% RSLogix 500 project vendingmachine.RSS, saved by version 9.00.00.04 %
PROJECT "UNTITLED"    % processor: MicroLogix 1200 %

PROGRAM FILES
  LAD 2   11 rungs

DATA FILES
  O0 OUTPUT  4 elements
  I1 INPUT  4 elements
  S2 STATUS  66 elements
  B3 BINARY  1 elements
  T4 TIMER  1 elements
  C5 COUNTER  1 elements
  R6 CONTROL  1 elements
  N7 INTEGER  1 elements
  F8 FLOAT  2 elements
  F9 PRICES  1 elements

LADDER 2
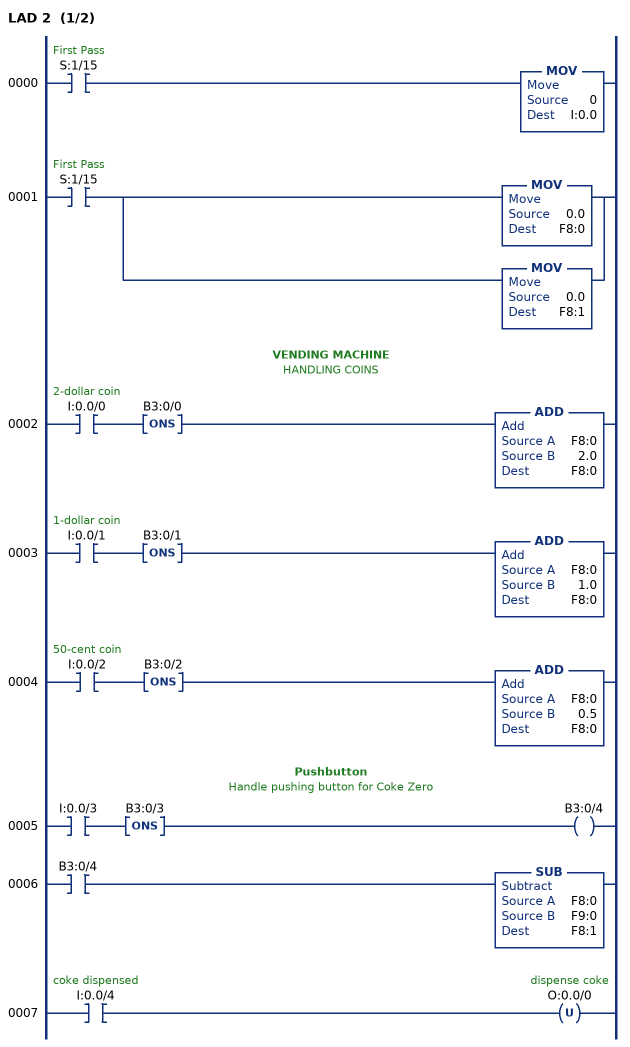
% Rung: 0 %
SOR XIC S:1/15 MOV 0 I:0.0 EOR
%   S:1/15  "First Pass" %
% Rung: 1 %
SOR XIC S:1/15 BST MOV 0.0 F8:0 NXB MOV 0.0 F8:1 BND EOR
%   S:1/15  "First Pass" %
% Rung: 2 %
% TITLE: VENDING MACHINE %
%                                                            HANDLING COINS %
SOR XIC I:0.0/0 ONS B3:0/0 ADD F8:0 2.0 F8:0 EOR
%   I:0.0/0  "2-dollar coin" %
% Rung: 3 %
SOR XIC I:0.0/1 ONS B3:0/1 ADD F8:0 1.0 F8:0 EOR
%   I:0.0/1  "1-dollar coin" %
% Rung: 4 %
SOR XIC I:0.0/2 ONS B3:0/2 ADD F8:0 0.5 F8:0 EOR
%   I:0.0/2  "50-cent coin" %
% Rung: 5 %
% TITLE: Pushbutton %
% Handle pushing button for Coke Zero %
SOR XIC I:0.0/3 ONS B3:0/3 OTE B3:0/4 EOR
% Rung: 6 %
SOR XIC B3:0/4 SUB F8:0 F9:0 F8:1 EOR
% Rung: 7 %
SOR XIC I:0.0/4 OTU O:0.0/0 EOR
%   I:0.0/4  "coke dispensed" %
%   O:0.0/0  "dispense coke" %

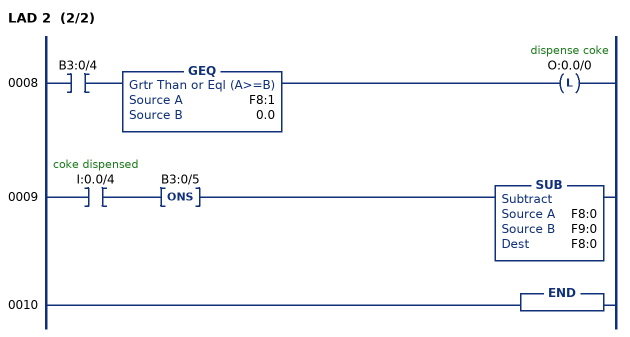
% Rung: 8 %
SOR XIC B3:0/4 GEQ F8:1 0.0 OTL O:0.0/0 EOR
%   O:0.0/0  "dispense coke" %
% Rung: 9 %
SOR XIC I:0.0/4 ONS B3:0/5 SUB F8:0 F9:0 F8:0 EOR
%   I:0.0/4  "coke dispensed" %
% Rung: 10 %
SOR END EOR

DATA TABLE (non-zero values as saved)
DATA B3
% B3:0 % 0X0008
DATA F9
% F9:0 % 2
